# EPICS autosave request: iocBoot/iocas/auto_positions.req
$(P)sample_positioner.VAL
